// Mitsubishi GX Developer project: 13-403_OLD_STyle   PLC: FX1S

PROGRAM MAIN
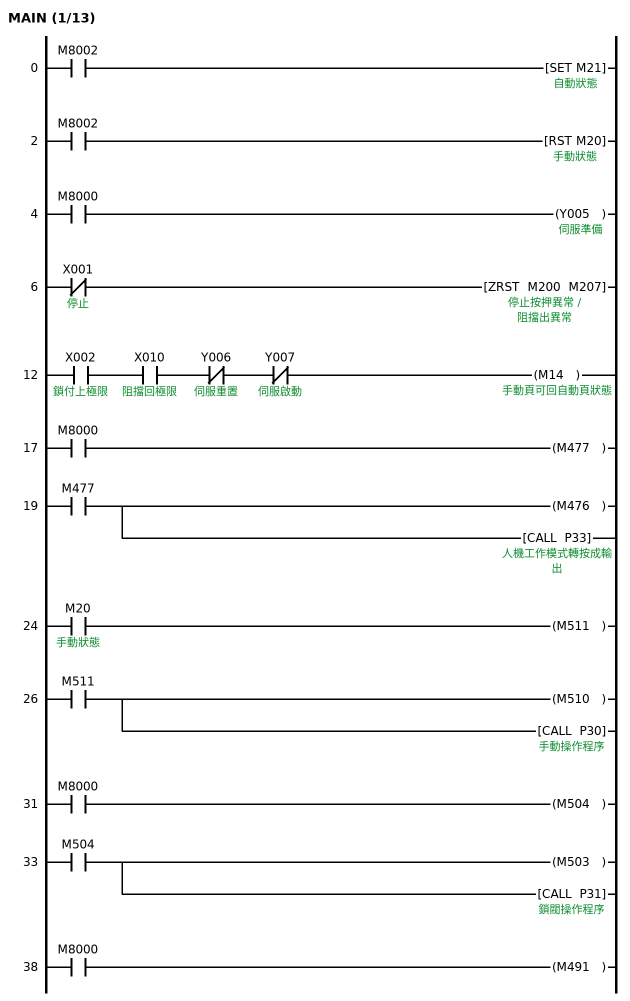
0     LD      M8002
      SET     M21  ; 自動狀態
2     LD      M8002
      RST     M20  ; 手動狀態
4     LD      M8000
      OUT     Y005  ; 伺服準備
6     LDI     X001  ; 停止
      ZRST    M200 M207  ; 停止按押異常 / 阻擋出異常
12    LD      X002  ; 鎖付上極限
      AND     X010  ; 阻擋回極限
      ANI     Y006  ; 伺服重置
      ANI     Y007  ; 伺服啟動
      OUT     M14  ; 手動頁可回自動頁狀態
17    LD      M8000
      OUT     M477
19    LD      M477
      OUT     M476
      CALL    P33  ; 人機工作模式轉按成輸出
24    LD      M20  ; 手動狀態
      OUT     M511
26    LD      M511
      OUT     M510
      CALL    P30  ; 手動操作程序
31    LD      M8000
      OUT     M504
33    LD      M504
      OUT     M503
      CALL    P31  ; 鎖閥操作程序
38    LD      M8000
      OUT     M491
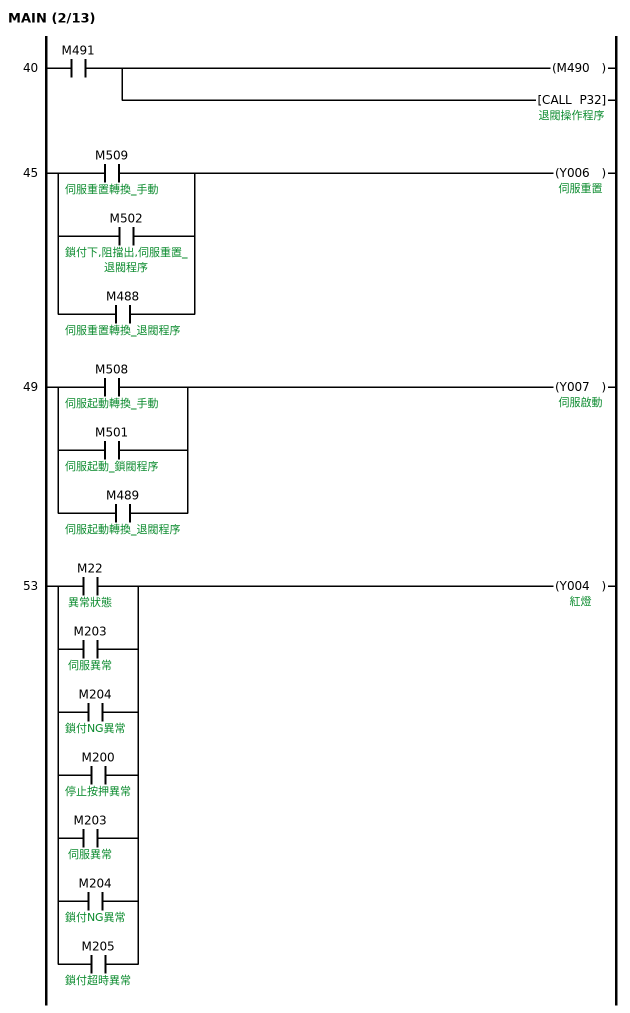
40    LD      M491
      OUT     M490
      CALL    P32  ; 退閥操作程序
45    LD      M509  ; 伺服重置轉換_手動
      OR      M502  ; 鎖付下,阻擋出,伺服重置_退閥程序
      OR      M488  ; 伺服重置轉換_退閥程序
      OUT     Y006  ; 伺服重置
49    LD      M508  ; 伺服起動轉換_手動
      OR      M501  ; 伺服起動_鎖閥程序
      OR      M489  ; 伺服起動轉換_退閥程序
      OUT     Y007  ; 伺服啟動
53    LD      M22  ; 異常狀態
      OR      M203  ; 伺服異常
      OR      M204  ; 鎖付NG異常
      OR      M200  ; 停止按押異常
      OR      M203  ; 伺服異常
      OR      M204  ; 鎖付NG異常
      OR      M205  ; 鎖付超時異常
      OUT     Y004  ; 紅燈
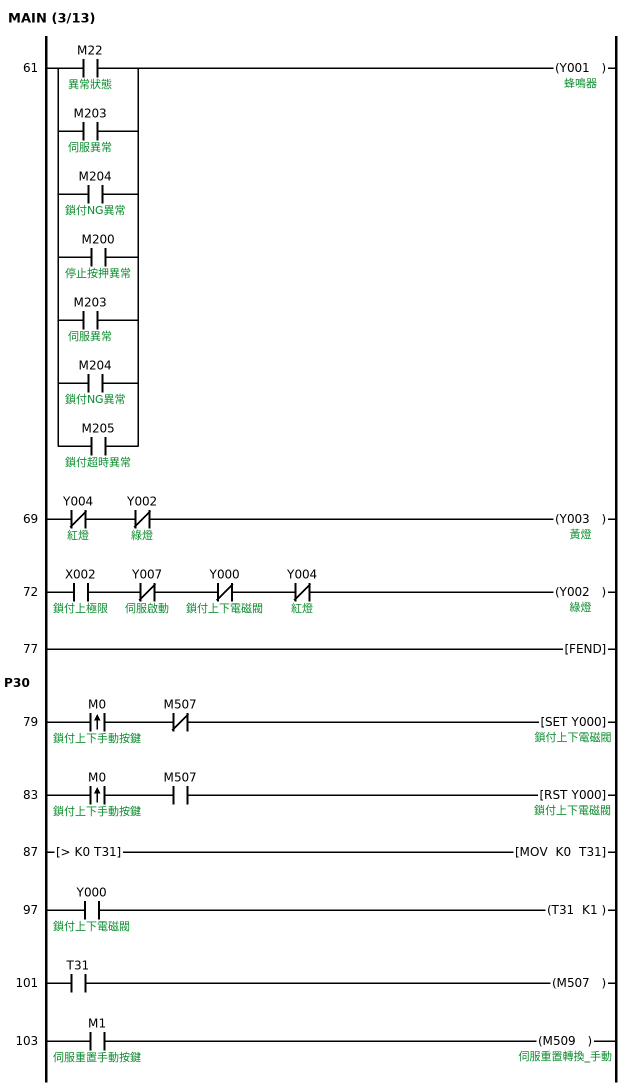
61    LD      M22  ; 異常狀態
      OR      M203  ; 伺服異常
      OR      M204  ; 鎖付NG異常
      OR      M200  ; 停止按押異常
      OR      M203  ; 伺服異常
      OR      M204  ; 鎖付NG異常
      OR      M205  ; 鎖付超時異常
      OUT     Y001  ; 蜂鳴器
69    LDI     Y004  ; 紅燈
      ANI     Y002  ; 綠燈
      OUT     Y003  ; 黃燈
72    LD      X002  ; 鎖付上極限
      ANI     Y007  ; 伺服啟動
      ANI     Y000  ; 鎖付上下電磁閥
      ANI     Y004  ; 紅燈
      OUT     Y002  ; 綠燈
77    FEND
      P30
79    LDP     M0  ; 鎖付上下手動按鍵
      ANI     M507
      SET     Y000  ; 鎖付上下電磁閥
83    LDP     M0  ; 鎖付上下手動按鍵
      AND     M507
      RST     Y000  ; 鎖付上下電磁閥
87    LD>     K0 T31
      MOV     K0 T31
97    LD      Y000  ; 鎖付上下電磁閥
      OUT     T31 K1
101   LD      T31
      OUT     M507
103   LD      M1  ; 伺服重置手動按鍵
      OUT     M509  ; 伺服重置轉換_手動
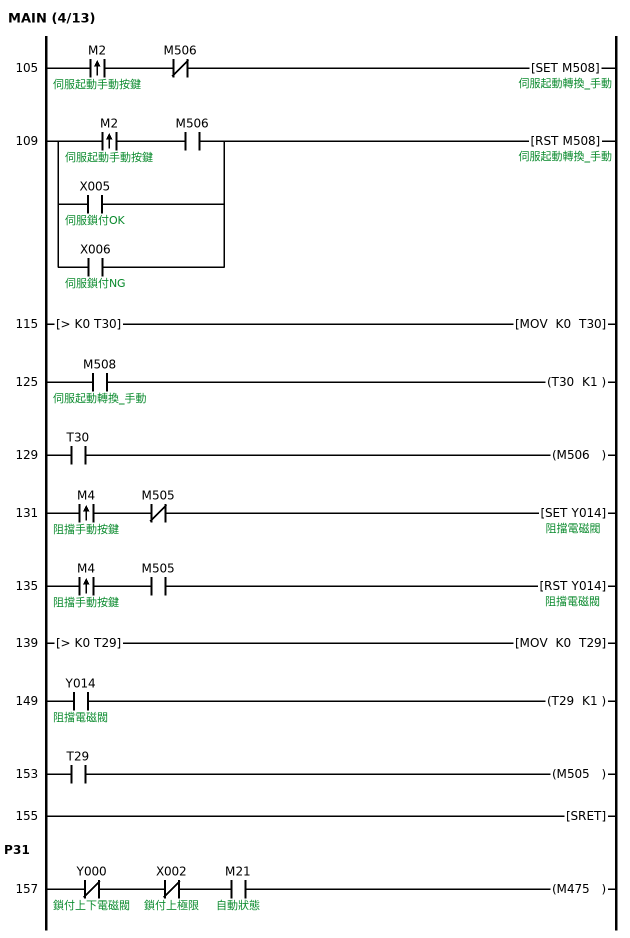
105   LDP     M2  ; 伺服起動手動按鍵
      ANI     M506
      SET     M508  ; 伺服起動轉換_手動
109   LDP     M2  ; 伺服起動手動按鍵
      AND     M506
      OR      X005  ; 伺服鎖付OK
      OR      X006  ; 伺服鎖付NG
      RST     M508  ; 伺服起動轉換_手動
115   LD>     K0 T30
      MOV     K0 T30
125   LD      M508  ; 伺服起動轉換_手動
      OUT     T30 K1
129   LD      T30
      OUT     M506
131   LDP     M4  ; 阻擋手動按鍵
      ANI     M505
      SET     Y014  ; 阻擋電磁閥
135   LDP     M4  ; 阻擋手動按鍵
      AND     M505
      RST     Y014  ; 阻擋電磁閥
139   LD>     K0 T29
      MOV     K0 T29
149   LD      Y014  ; 阻擋電磁閥
      OUT     T29 K1
153   LD      T29
      OUT     M505
155   SRET
      P31
157   LDI     Y000  ; 鎖付上下電磁閥
      ANI     X002  ; 鎖付上極限
      AND     M21  ; 自動狀態
      OUT     M475
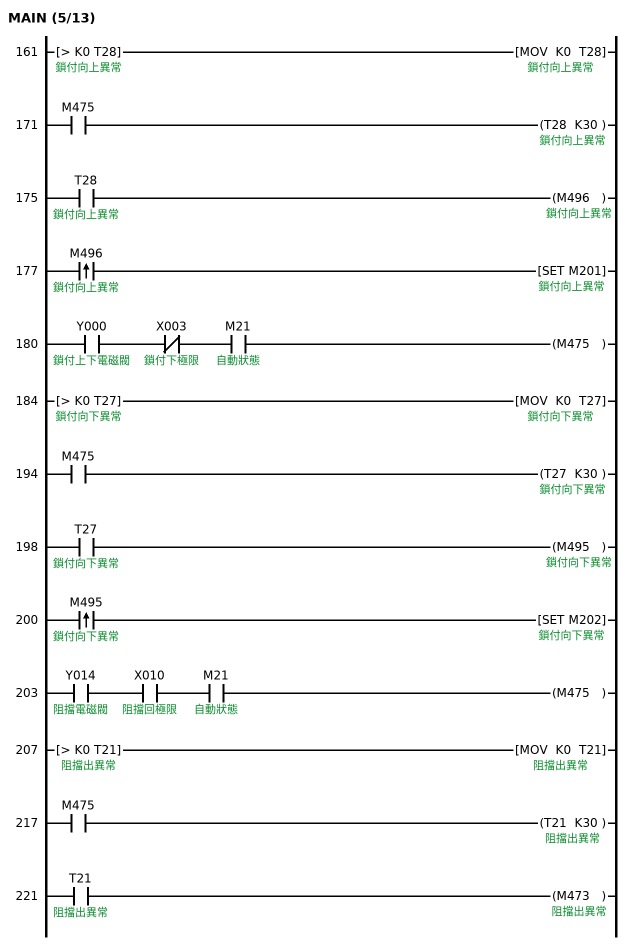
161   LD>     K0 T28  ; 鎖付向上異常
      MOV     K0 T28
171   LD      M475
      OUT     T28 K30  ; 鎖付向上異常
175   LD      T28  ; 鎖付向上異常
      OUT     M496  ; 鎖付向上異常
177   LDP     M496  ; 鎖付向上異常
      SET     M201  ; 鎖付向上異常
180   LD      Y000  ; 鎖付上下電磁閥
      ANI     X003  ; 鎖付下極限
      AND     M21  ; 自動狀態
      OUT     M475
184   LD>     K0 T27  ; 鎖付向下異常
      MOV     K0 T27
194   LD      M475
      OUT     T27 K30  ; 鎖付向下異常
198   LD      T27  ; 鎖付向下異常
      OUT     M495  ; 鎖付向下異常
200   LDP     M495  ; 鎖付向下異常
      SET     M202  ; 鎖付向下異常
203   LD      Y014  ; 阻擋電磁閥
      AND     X010  ; 阻擋回極限
      AND     M21  ; 自動狀態
      OUT     M475
207   LD>     K0 T21  ; 阻擋出異常
      MOV     K0 T21
217   LD      M475
      OUT     T21 K30  ; 阻擋出異常
221   LD      T21  ; 阻擋出異常
      OUT     M473  ; 阻擋出異常
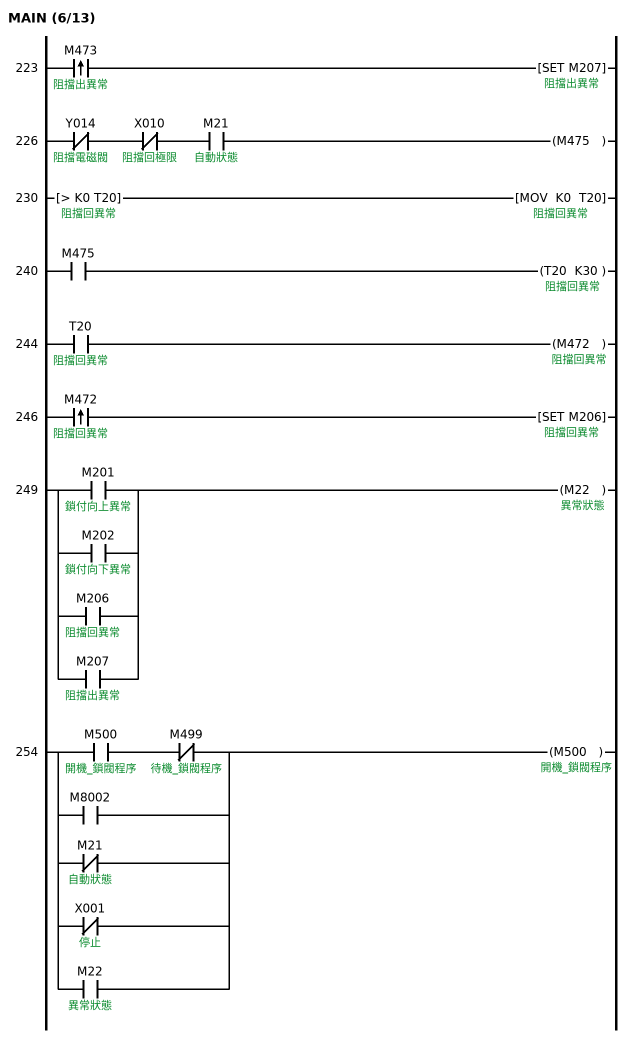
223   LDP     M473  ; 阻擋出異常
      SET     M207  ; 阻擋出異常
226   LDI     Y014  ; 阻擋電磁閥
      ANI     X010  ; 阻擋回極限
      AND     M21  ; 自動狀態
      OUT     M475
230   LD>     K0 T20  ; 阻擋回異常
      MOV     K0 T20
240   LD      M475
      OUT     T20 K30  ; 阻擋回異常
244   LD      T20  ; 阻擋回異常
      OUT     M472  ; 阻擋回異常
246   LDP     M472  ; 阻擋回異常
      SET     M206  ; 阻擋回異常
249   LD      M201  ; 鎖付向上異常
      OR      M202  ; 鎖付向下異常
      OR      M206  ; 阻擋回異常
      OR      M207  ; 阻擋出異常
      OUT     M22  ; 異常狀態
254   LD      M500  ; 開機_鎖閥程序
      ANI     M499  ; 待機_鎖閥程序
      OR      M8002
      ORI     M21  ; 自動狀態
      ORI     X001  ; 停止
      OR      M22  ; 異常狀態
      OUT     M500  ; 開機_鎖閥程序
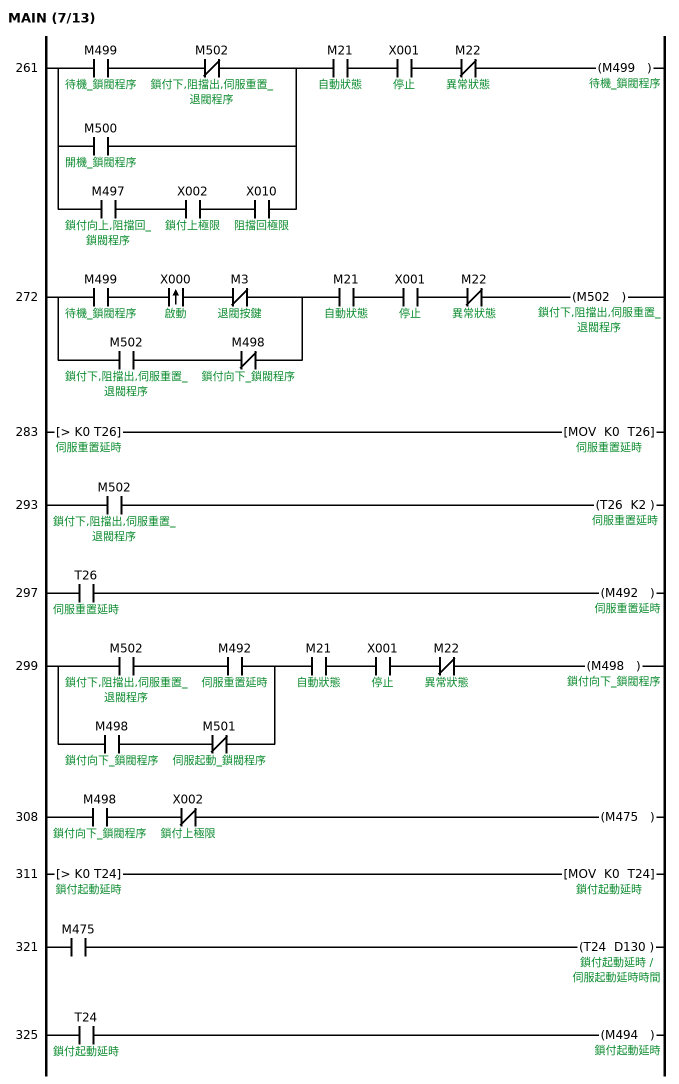
261   LD      M499  ; 待機_鎖閥程序
      ANI     M502  ; 鎖付下,阻擋出,伺服重置_退閥程序
      OR      M500  ; 開機_鎖閥程序
      LD      M497  ; 鎖付向上,阻擋回_鎖閥程序
      AND     X002  ; 鎖付上極限
      AND     X010  ; 阻擋回極限
      ORB
      AND     M21  ; 自動狀態
      AND     X001  ; 停止
      ANI     M22  ; 異常狀態
      OUT     M499  ; 待機_鎖閥程序
272   LD      M499  ; 待機_鎖閥程序
      ANDP    X000  ; 啟動
      ANI     M3  ; 退閥按鍵
      LD      M502  ; 鎖付下,阻擋出,伺服重置_退閥程序
      ANI     M498  ; 鎖付向下_鎖閥程序
      ORB
      AND     M21  ; 自動狀態
      AND     X001  ; 停止
      ANI     M22  ; 異常狀態
      OUT     M502  ; 鎖付下,阻擋出,伺服重置_退閥程序
283   LD>     K0 T26  ; 伺服重置延時
      MOV     K0 T26
293   LD      M502  ; 鎖付下,阻擋出,伺服重置_退閥程序
      OUT     T26 K2  ; 伺服重置延時
297   LD      T26  ; 伺服重置延時
      OUT     M492  ; 伺服重置延時
299   LD      M502  ; 鎖付下,阻擋出,伺服重置_退閥程序
      AND     M492  ; 伺服重置延時
      LD      M498  ; 鎖付向下_鎖閥程序
      ANI     M501  ; 伺服起動_鎖閥程序
      ORB
      AND     M21  ; 自動狀態
      AND     X001  ; 停止
      ANI     M22  ; 異常狀態
      OUT     M498  ; 鎖付向下_鎖閥程序
308   LD      M498  ; 鎖付向下_鎖閥程序
      ANI     X002  ; 鎖付上極限
      OUT     M475
311   LD>     K0 T24  ; 鎖付起動延時
      MOV     K0 T24
321   LD      M475
      OUT     T24 D130  ; 鎖付起動延時 / 伺服起動延時時間
325   LD      T24  ; 鎖付起動延時
      OUT     M494  ; 鎖付起動延時
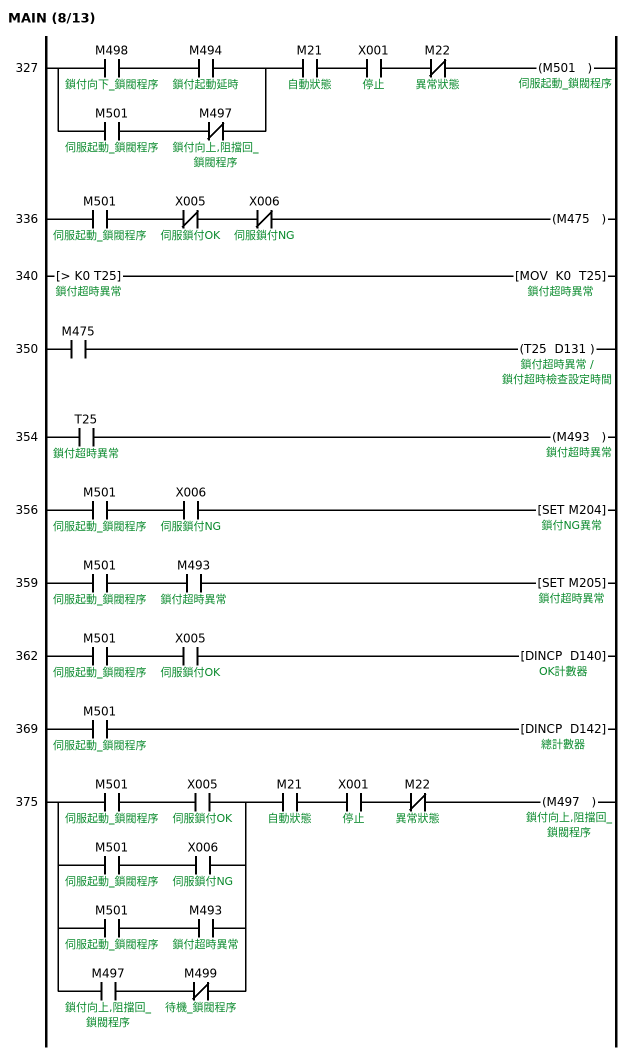
327   LD      M498  ; 鎖付向下_鎖閥程序
      AND     M494  ; 鎖付起動延時
      LD      M501  ; 伺服起動_鎖閥程序
      ANI     M497  ; 鎖付向上,阻擋回_鎖閥程序
      ORB
      AND     M21  ; 自動狀態
      AND     X001  ; 停止
      ANI     M22  ; 異常狀態
      OUT     M501  ; 伺服起動_鎖閥程序
336   LD      M501  ; 伺服起動_鎖閥程序
      ANI     X005  ; 伺服鎖付OK
      ANI     X006  ; 伺服鎖付NG
      OUT     M475
340   LD>     K0 T25  ; 鎖付超時異常
      MOV     K0 T25
350   LD      M475
      OUT     T25 D131  ; 鎖付超時異常 / 鎖付超時檢查設定時間
354   LD      T25  ; 鎖付超時異常
      OUT     M493  ; 鎖付超時異常
356   LD      M501  ; 伺服起動_鎖閥程序
      AND     X006  ; 伺服鎖付NG
      SET     M204  ; 鎖付NG異常
359   LD      M501  ; 伺服起動_鎖閥程序
      AND     M493  ; 鎖付超時異常
      SET     M205  ; 鎖付超時異常
362   LD      M501  ; 伺服起動_鎖閥程序
      AND     X005  ; 伺服鎖付OK
      DINCP   D140  ; OK計數器
369   LD      M501  ; 伺服起動_鎖閥程序
      DINCP   D142  ; 總計數器
375   LD      M501  ; 伺服起動_鎖閥程序
      AND     X005  ; 伺服鎖付OK
      LD      M501  ; 伺服起動_鎖閥程序
      AND     X006  ; 伺服鎖付NG
      ORB
      LD      M501  ; 伺服起動_鎖閥程序
      AND     M493  ; 鎖付超時異常
      ORB
      LD      M497  ; 鎖付向上,阻擋回_鎖閥程序
      ANI     M499  ; 待機_鎖閥程序
      ORB
      AND     M21  ; 自動狀態
      AND     X001  ; 停止
      ANI     M22  ; 異常狀態
      OUT     M497  ; 鎖付向上,阻擋回_鎖閥程序
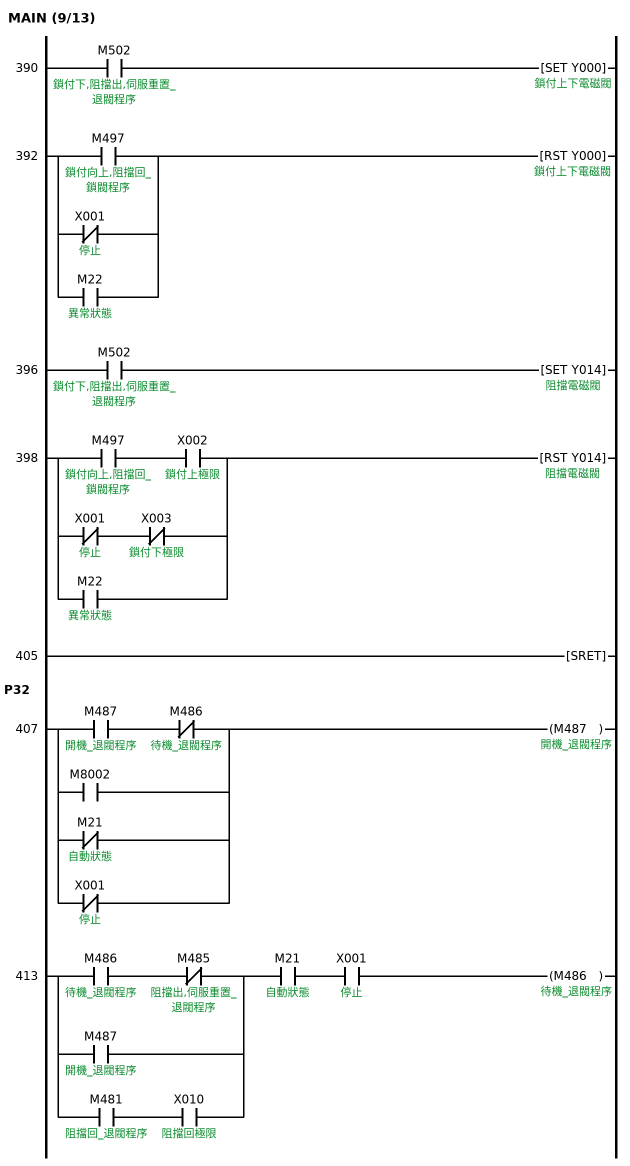
390   LD      M502  ; 鎖付下,阻擋出,伺服重置_退閥程序
      SET     Y000  ; 鎖付上下電磁閥
392   LD      M497  ; 鎖付向上,阻擋回_鎖閥程序
      ORI     X001  ; 停止
      OR      M22  ; 異常狀態
      RST     Y000  ; 鎖付上下電磁閥
396   LD      M502  ; 鎖付下,阻擋出,伺服重置_退閥程序
      SET     Y014  ; 阻擋電磁閥
398   LD      M497  ; 鎖付向上,阻擋回_鎖閥程序
      AND     X002  ; 鎖付上極限
      LDI     X001  ; 停止
      ANI     X003  ; 鎖付下極限
      ORB
      OR      M22  ; 異常狀態
      RST     Y014  ; 阻擋電磁閥
405   SRET
      P32
407   LD      M487  ; 開機_退閥程序
      ANI     M486  ; 待機_退閥程序
      OR      M8002
      ORI     M21  ; 自動狀態
      ORI     X001  ; 停止
      OUT     M487  ; 開機_退閥程序
413   LD      M486  ; 待機_退閥程序
      ANI     M485  ; 阻擋出,伺服重置_退閥程序
      OR      M487  ; 開機_退閥程序
      LD      M481  ; 阻擋回_退閥程序
      AND     X010  ; 阻擋回極限
      ORB
      AND     M21  ; 自動狀態
      AND     X001  ; 停止
      OUT     M486  ; 待機_退閥程序
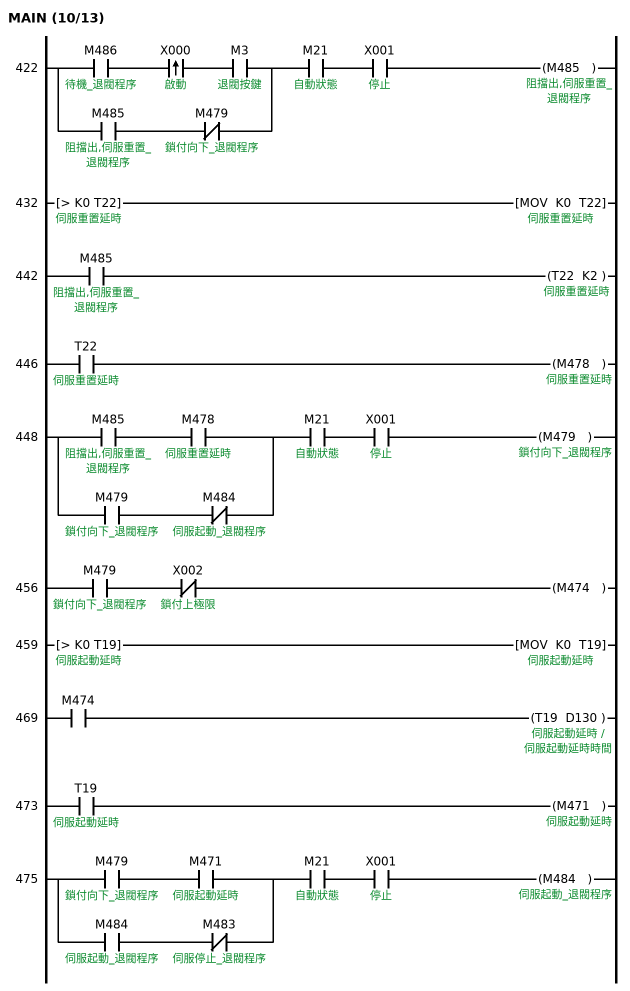
422   LD      M486  ; 待機_退閥程序
      ANDP    X000  ; 啟動
      AND     M3  ; 退閥按鍵
      LD      M485  ; 阻擋出,伺服重置_退閥程序
      ANI     M479  ; 鎖付向下_退閥程序
      ORB
      AND     M21  ; 自動狀態
      AND     X001  ; 停止
      OUT     M485  ; 阻擋出,伺服重置_退閥程序
432   LD>     K0 T22  ; 伺服重置延時
      MOV     K0 T22
442   LD      M485  ; 阻擋出,伺服重置_退閥程序
      OUT     T22 K2  ; 伺服重置延時
446   LD      T22  ; 伺服重置延時
      OUT     M478  ; 伺服重置延時
448   LD      M485  ; 阻擋出,伺服重置_退閥程序
      AND     M478  ; 伺服重置延時
      LD      M479  ; 鎖付向下_退閥程序
      ANI     M484  ; 伺服起動_退閥程序
      ORB
      AND     M21  ; 自動狀態
      AND     X001  ; 停止
      OUT     M479  ; 鎖付向下_退閥程序
456   LD      M479  ; 鎖付向下_退閥程序
      ANI     X002  ; 鎖付上極限
      OUT     M474
459   LD>     K0 T19  ; 伺服起動延時
      MOV     K0 T19
469   LD      M474
      OUT     T19 D130  ; 伺服起動延時 / 伺服起動延時時間
473   LD      T19  ; 伺服起動延時
      OUT     M471  ; 伺服起動延時
475   LD      M479  ; 鎖付向下_退閥程序
      AND     M471  ; 伺服起動延時
      LD      M484  ; 伺服起動_退閥程序
      ANI     M483  ; 伺服停止_退閥程序
      ORB
      AND     M21  ; 自動狀態
      AND     X001  ; 停止
      OUT     M484  ; 伺服起動_退閥程序
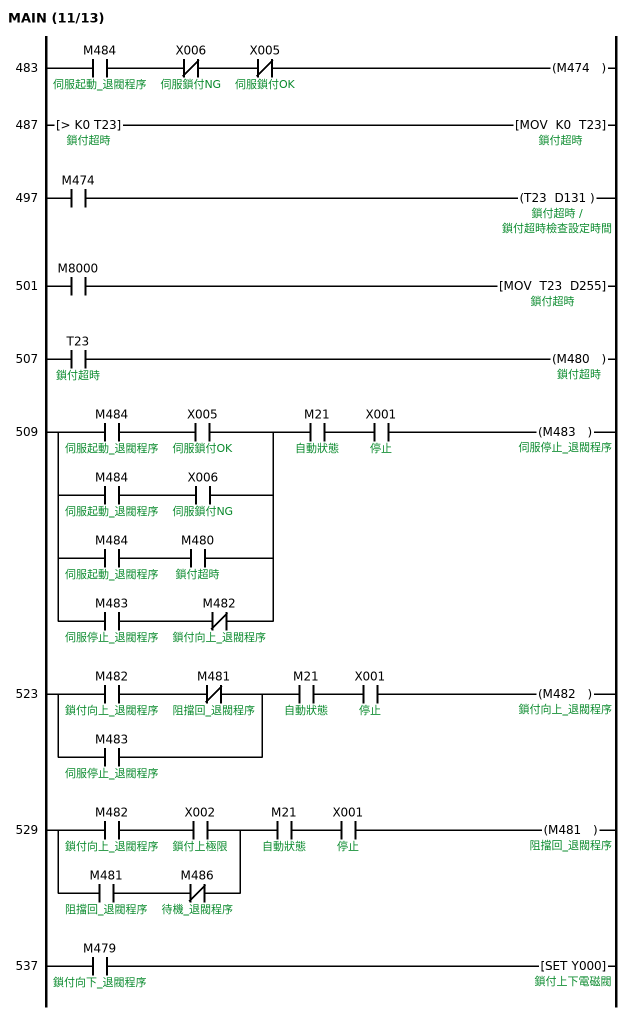
483   LD      M484  ; 伺服起動_退閥程序
      ANI     X006  ; 伺服鎖付NG
      ANI     X005  ; 伺服鎖付OK
      OUT     M474
487   LD>     K0 T23  ; 鎖付超時
      MOV     K0 T23
497   LD      M474
      OUT     T23 D131  ; 鎖付超時 / 鎖付超時檢查設定時間
501   LD      M8000
      MOV     T23 D255
507   LD      T23  ; 鎖付超時
      OUT     M480  ; 鎖付超時
509   LD      M484  ; 伺服起動_退閥程序
      AND     X005  ; 伺服鎖付OK
      LD      M484  ; 伺服起動_退閥程序
      AND     X006  ; 伺服鎖付NG
      ORB
      LD      M484  ; 伺服起動_退閥程序
      AND     M480  ; 鎖付超時
      ORB
      LD      M483  ; 伺服停止_退閥程序
      ANI     M482  ; 鎖付向上_退閥程序
      ORB
      AND     M21  ; 自動狀態
      AND     X001  ; 停止
      OUT     M483  ; 伺服停止_退閥程序
523   LD      M482  ; 鎖付向上_退閥程序
      ANI     M481  ; 阻擋回_退閥程序
      OR      M483  ; 伺服停止_退閥程序
      AND     M21  ; 自動狀態
      AND     X001  ; 停止
      OUT     M482  ; 鎖付向上_退閥程序
529   LD      M482  ; 鎖付向上_退閥程序
      AND     X002  ; 鎖付上極限
      LD      M481  ; 阻擋回_退閥程序
      ANI     M486  ; 待機_退閥程序
      ORB
      AND     M21  ; 自動狀態
      AND     X001  ; 停止
      OUT     M481  ; 阻擋回_退閥程序
537   LD      M479  ; 鎖付向下_退閥程序
      SET     Y000  ; 鎖付上下電磁閥
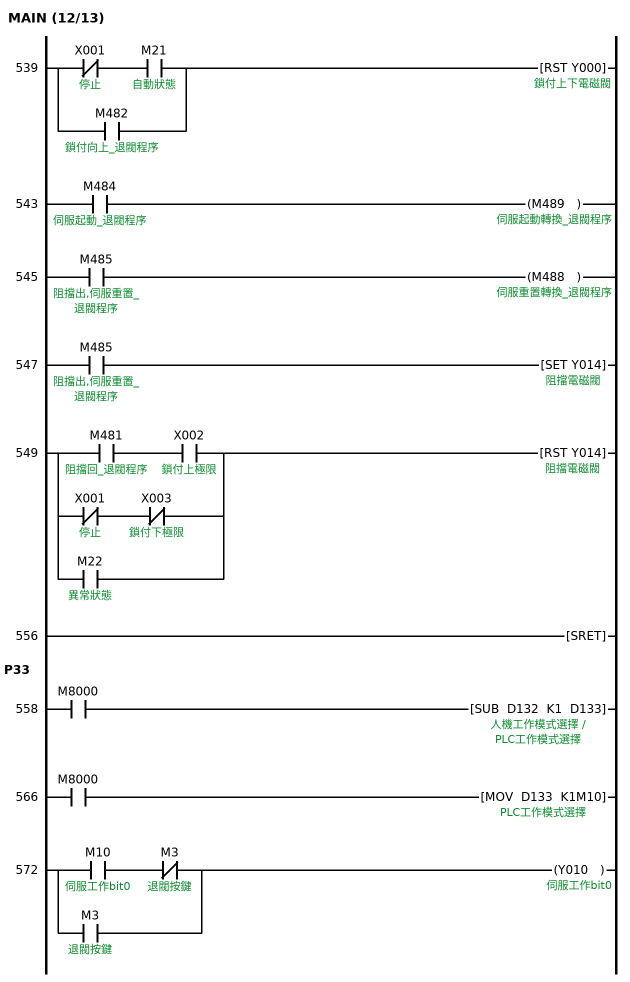
539   LDI     X001  ; 停止
      AND     M21  ; 自動狀態
      OR      M482  ; 鎖付向上_退閥程序
      RST     Y000  ; 鎖付上下電磁閥
543   LD      M484  ; 伺服起動_退閥程序
      OUT     M489  ; 伺服起動轉換_退閥程序
545   LD      M485  ; 阻擋出,伺服重置_退閥程序
      OUT     M488  ; 伺服重置轉換_退閥程序
547   LD      M485  ; 阻擋出,伺服重置_退閥程序
      SET     Y014  ; 阻擋電磁閥
549   LD      M481  ; 阻擋回_退閥程序
      AND     X002  ; 鎖付上極限
      LDI     X001  ; 停止
      ANI     X003  ; 鎖付下極限
      ORB
      OR      M22  ; 異常狀態
      RST     Y014  ; 阻擋電磁閥
556   SRET
      P33
558   LD      M8000
      SUB     D132 K1 D133  ; 人機工作模式選擇 / PLC工作模式選擇
566   LD      M8000
      MOV     D133 K1M10  ; 伺服工作bit0
572   LD      M10  ; 伺服工作bit0
      ANI     M3  ; 退閥按鍵
      OR      M3  ; 退閥按鍵
      OUT     Y010  ; 伺服工作bit0
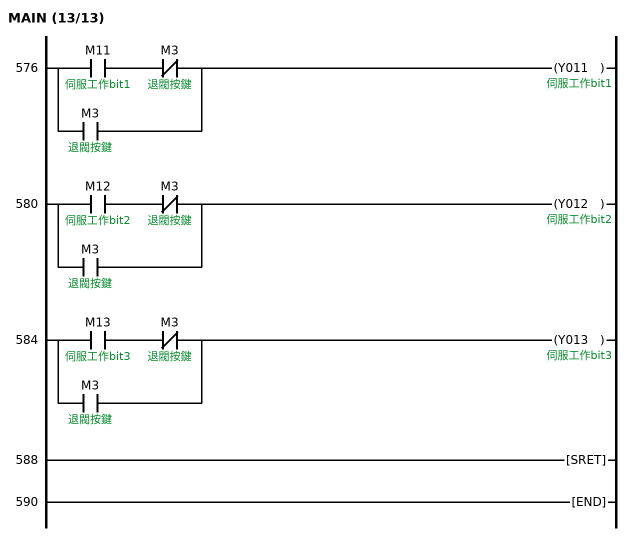
576   LD      M11  ; 伺服工作bit1
      ANI     M3  ; 退閥按鍵
      OR      M3  ; 退閥按鍵
      OUT     Y011  ; 伺服工作bit1
580   LD      M12  ; 伺服工作bit2
      ANI     M3  ; 退閥按鍵
      OR      M3  ; 退閥按鍵
      OUT     Y012  ; 伺服工作bit2
584   LD      M13  ; 伺服工作bit3
      ANI     M3  ; 退閥按鍵
      OR      M3  ; 退閥按鍵
      OUT     Y013  ; 伺服工作bit3
588   SRET
590   END
END_PROGRAM

// device comments not shown above
X004  ; 伺服異常
D141  ; *************
D143  ; *************
